// Mitsubishi GX Works2 project: solar   PLC: FX3U/FX3UC

PROGRAM MAIN
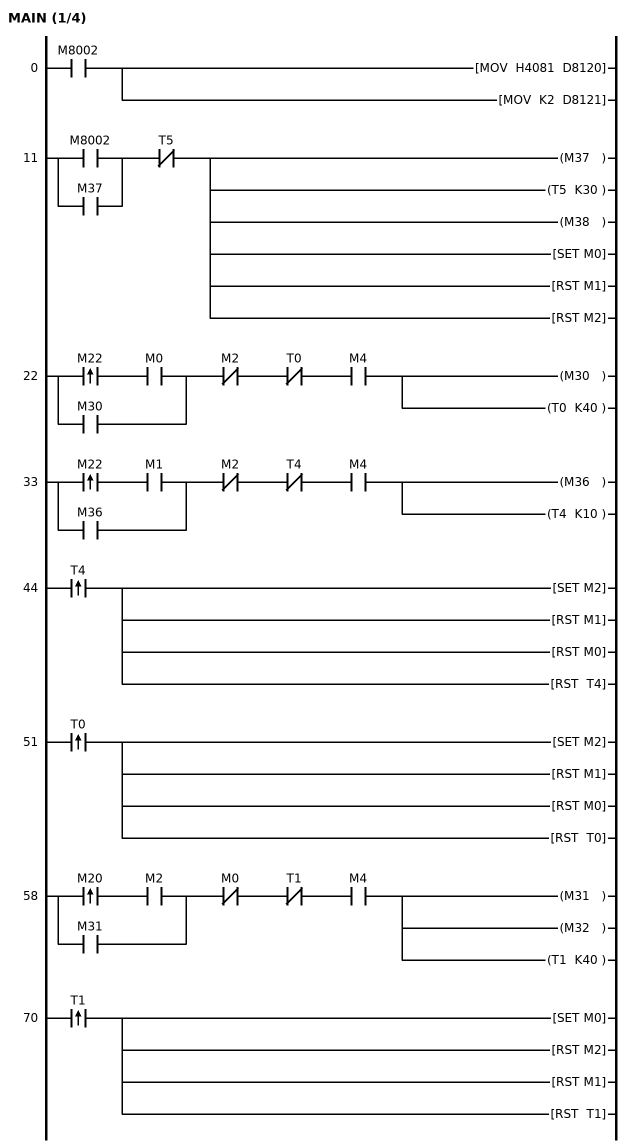
0     LD      M8002
      MOV     H4081 D8120
      MOV     K2 D8121
11    LD      M8002
      OR      M37
      ANI     T5
      OUT     M37
      OUT     T5 K30
      OUT     M38
      SET     M0
      RST     M1
      RST     M2
22    LDP     M22
      AND     M0
      OR      M30
      ANI     M2
      ANI     T0
      AND     M4
      OUT     M30
      OUT     T0 K40
33    LDP     M22
      AND     M1
      OR      M36
      ANI     M2
      ANI     T4
      AND     M4
      OUT     M36
      OUT     T4 K10
44    LDP     T4
      SET     M2
      RST     M1
      RST     M0
      RST     T4
51    LDP     T0
      SET     M2
      RST     M1
      RST     M0
      RST     T0
58    LDP     M20
      AND     M2
      OR      M31
      ANI     M0
      ANI     T1
      AND     M4
      OUT     M31
      OUT     M32
      OUT     T1 K40
70    LDP     T1
      SET     M0
      RST     M2
      RST     M1
      RST     T1
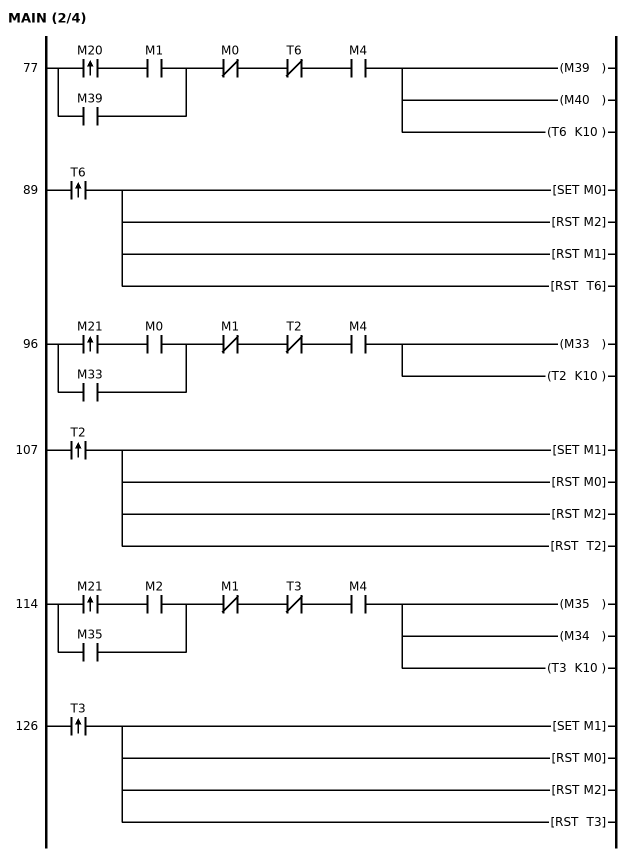
77    LDP     M20
      AND     M1
      OR      M39
      ANI     M0
      ANI     T6
      AND     M4
      OUT     M39
      OUT     M40
      OUT     T6 K10
89    LDP     T6
      SET     M0
      RST     M2
      RST     M1
      RST     T6
96    LDP     M21
      AND     M0
      OR      M33
      ANI     M1
      ANI     T2
      AND     M4
      OUT     M33
      OUT     T2 K10
107   LDP     T2
      SET     M1
      RST     M0
      RST     M2
      RST     T2
114   LDP     M21
      AND     M2
      OR      M35
      ANI     M1
      ANI     T3
      AND     M4
      OUT     M35
      OUT     M34
      OUT     T3 K10
126   LDP     T3
      SET     M1
      RST     M0
      RST     M2
      RST     T3
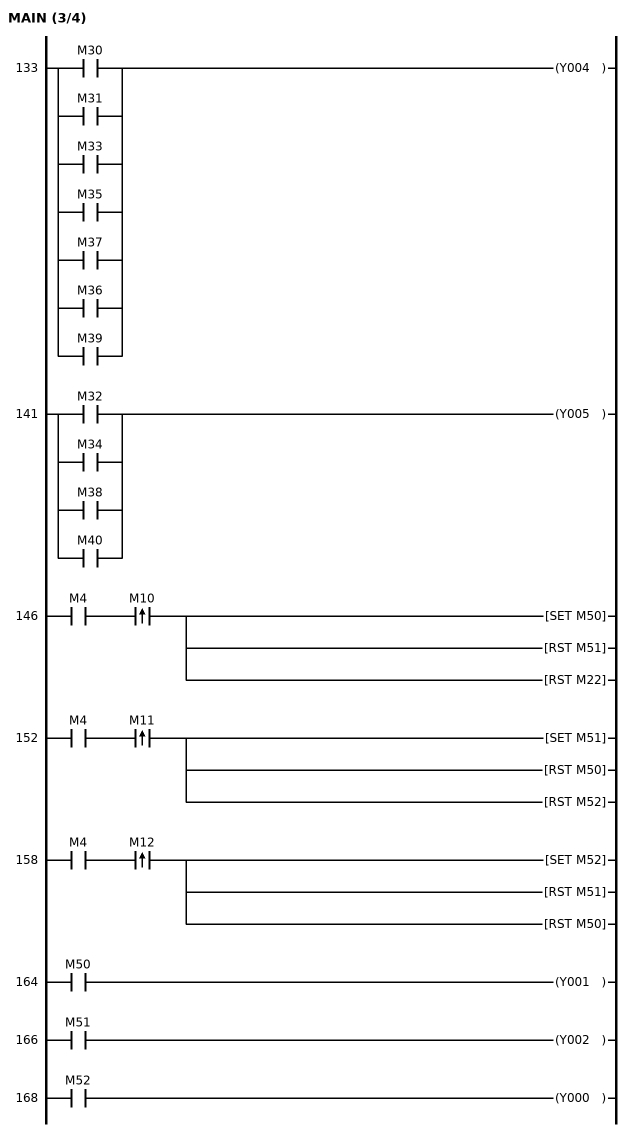
133   LD      M30
      OR      M31
      OR      M33
      OR      M35
      OR      M37
      OR      M36
      OR      M39
      OUT     Y004
141   LD      M32
      OR      M34
      OR      M38
      OR      M40
      OUT     Y005
146   LD      M4
      ANDP    M10
      SET     M50
      RST     M51
      RST     M22
152   LD      M4
      ANDP    M11
      SET     M51
      RST     M50
      RST     M52
158   LD      M4
      ANDP    M12
      SET     M52
      RST     M51
      RST     M50
164   LD      M50
      OUT     Y001
166   LD      M51
      OUT     Y002
168   LD      M52
      OUT     Y000
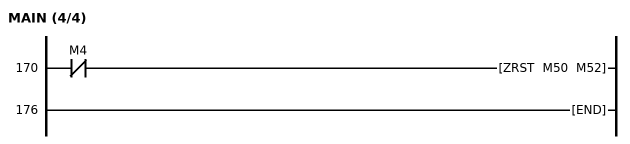
170   LDI     M4
      ZRST    M50 M52
176   END
END_PROGRAM
